(* IEC 61131-3 sources: test/Class/SfcClass_Action0, 1 file *)

(* ---- SfcClass_Action0.st ---- *)
(*!
<Class
	Name               = "SfcClass_Action0"
	Revision           = "0.0"
	RealtimeTask       = "false"
	CyclicTask         = "false"
	BackgroundTask     = "false"
	Sigmatek           = "false"
	OSInterface        = "false"
	HighPriority       = "false"
	Automatic          = "false"
	UpdateMode         = "Prescan"
	SharedCommandTable = "true"
	Objectsize         = "(284,120)">
	<Channels>
	</Channels>
	<Network Name="SfcClass_Action0">
		<!-- List of Components in this network -->
		<Components>
			<Object
				Name       = "_base"
				Class      = "Sfc_Action_Base"
				Position   = "(218,120)"
				Visualized = "true"
				Remotely   = "true">
				<Channels>
					<Server Name="A"/>
					<Server Name="DelayActive"/>
					<Server Name="Itf"/>
					<Server Name="Q"/>
					<Server Name="T"/>
					<Client Name="GetParentPtr"/>
					<Client Name="LogonToInvoker"/>
				</Channels>
			</Object>
		</Components>
		<Comments>
		</Comments>
		<!-- List of Connections in this network -->
		<Connections>
			<Connection Source="this.Itf" Destination="_base.Itf" Vertices="(690,210),(518,210),"/>
			<Connection Source="this.A" Destination="_base.A" Vertices="(690,270),(518,270),"/>
			<Connection Source="this.T" Destination="_base.T" Vertices="(690,330),(518,330),"/>
			<Connection Source="this.Q" Destination="_base.Q" Vertices="(690,390),(518,390),"/>
			<Connection Source="this.DelayActive" Destination="_base.DelayActive" Vertices="(690,450),(518,450),"/>
			<Connection Source="_base.LogonToInvoker" Destination="this.LogonToInvoker" Vertices="(230,210),(38,210),"/>
			<Connection Source="_base.GetParentPtr" Destination="this.GetParentPtr" Vertices="(230,270),(38,270),"/>
		</Connections>
		<!-- Headerfiles -->
		<Options>
		</Options>
	</Network>
</Class>
*)
#pragma using Sfc_Action_Base

SfcClass_Action0 : CLASS
: Sfc_Action_Base
	TYPE
	  pParentClsPtr : ^SfcClass;
	END_TYPE
  //Servers:
  //Clients:
  //Variables:
  //Functions:

	FUNCTION VIRTUAL OnWork;
				//! <Function Name="OnReadInternalVariables" Hidden="true"/>
	FUNCTION VIRTUAL OnReadInternalVariables;
				//! <Function Name="OnWriteInternalVariables" Hidden="true"/>
	FUNCTION VIRTUAL OnWriteInternalVariables;
  //Tables:
	FUNCTION @STD
		VAR_OUTPUT
			ret_code	: CONFSTATES;
		END_VAR;
	FUNCTION GLOBAL TAB @CT_;
END_CLASS;

#pragma usingLtd SfcClass

FUNCTION VIRTUAL SfcClass_Action0::OnReadInternalVariables

END_FUNCTION
FUNCTION VIRTUAL SfcClass_Action0::OnWriteInternalVariables

END_FUNCTION

FUNCTION VIRTUAL SfcClass_Action0::OnWork

END_FUNCTION
